{attribute 'qualified_only' := ''}
{attribute 'strict' := ''}
TYPE cPuckStatusEval :
(
	None := 0
) DINT;
END_TYPE

(* stored: Version 1.1.0.1, ProductVersion 3.1.4024.6
   DUT cPuckStatusEval: Id {878aa6be-cfc2-4e2c-8f51-1fde2a0c82d6} *)
